(* IEC 61131-3 sources: Industry-PLC-LLM/data/PLCBEAD_repo/PLCBEAD_PLCEmbed-main/PLC-BEAD/Source/GEB/DATE_TO_REAL, 1 file *)

(* ---- DATE_TO_REAL.ST ---- *)
FUNCTION DATE_TO_REAL2:REAL
	VAR_INPUT
		IN :	UDINT;
	END_VAR

	DATE_TO_REAL2 := UDINT_TO_REAL(IN);
END_FUNCTION

PROGRAM program0
  VAR
    LocalVar0 : UDINT;
	LocalOUT  : REAL;
  END_VAR
  	LocalOUT := DATE_TO_REAL2(LocalVar0);
END_PROGRAM
